PROGRAM P_WenglorTeach
VAR
	bTeachModeCapCheck:BOOL;
	bTeachModeCapCorrect:BOOL;
	tofTeachModeCapCheck:TOF;
	tofTeachModeCapCorrect:TOF;
	fbAverageValueCapCheck: FB_Average;
	fbAverageValueCapCorrect: FB_Average;
END_VAR

tofTeachModeCapCheck(IN:=bTeachModeCapCheck,PT:=T#10S);
tofTeachModeCapCorrect(IN:=bTeachModeCapCorrect,PT:=T#10S);
IF tofTeachModeCapCheck.q THEN
	fbAverageValueCapCheck(rValue:=LREAL_TO_REAL(P09_CapPuttedCheck.lrCapPuttedCheckSensorCV), tInterval:= T#5MS, rAverage=>);
END_IF
IF tofTeachModeCapCorrect.q THEN
	fbAverageValueCapCorrect(rValue:=LREAL_TO_REAL(P11_CapCorrectCheck.lrCapCorrectCheckSensorCV), tInterval:= T#5MS, rAverage=>);
END_IF

END_PROGRAM

(* stored: Version 1.1.0.1, ProductVersion 3.1.4026.13, FileIdentifier b87d97fcc3b6a8492774223f31377b2b3b25ad86, FileSignature 32f6c711464d3a500181e8f54a3465f7cfa7e3caf1fcd915abd1e3a4dd0e0a5eb8aab20f0863e098b1ceb5766523403dffb33ecec23c48b2d643c0c45e48e1e8898ed60869a301a0bdb07f630975f28fc0430427ac1f4a55742bd6d8dd972a58a18f1deda52c4cfe5d1a275f2011370d0037661f8dd59b43e51bd3034f9a9a1e0ea04ed72ffa408e7a8ff1874d29dc4a6fb24c46d5c88dd33c00516d3d9d6eb41f240d304061d6dc5a7c67965c51793dfa4158aee50363ca5a9c06c38d041dcd37c5fee7296248bf21f4554e4015d48503b402175ca859e306246e5881ca491d2854f8cb8479387f519b1eb44c781306def177cda3367bc8c1099f308cd13f5c
   POU P_WenglorTeach: Id {13c18d49-c970-45f2-8a1b-6c305bfd3563}, SpecialFunc None *)
